INTERFACE I_State

METHOD Disable : BOOL
VAR_INPUT
END_VAR
END_METHOD

METHOD Enable : BOOL
VAR_INPUT
END_VAR
END_METHOD

METHOD Reset : BOOL
VAR_INPUT
END_VAR
END_METHOD

END_INTERFACE

(* stored: Version 1.1.0.1, ProductVersion 3.1.4024.3
   Itf I_State: Id {531fa272-2cd5-42d8-9cf4-4c3ca4bd3b79}
   Method Disable: Id {1cfec2c5-39b9-4c11-9f5f-160761311480}
   Method Enable: Id {344e01c2-3887-49b7-8e4c-b1d7a2ec73ab}
   Method Reset: Id {38174c13-87a3-4d7f-8d74-3b6394874f7b} *)
